FUNCTION_BLOCK Clearing_State  IMPLEMENTS ITF_State
VAR_INPUT
END_VAR
VAR_OUTPUT
END_VAR
VAR
	pPML_Base : POINTER TO PML_StatePattern_Base;
	_stateMachine : IPmlStateMachine;
END_VAR

METHOD Cycle : BOOL
_stateMachine.SetStateComplete();
pPML_Base^.SetState(pPML_Base^.stopped);
END_METHOD

METHOD FB_init : BOOL
VAR_INPUT
	bInitRetains : BOOL; // if TRUE, the retain variables are initialized (warm start / cold start)
	bInCopyCode : BOOL;  // if TRUE, the instance afterwards gets moved into the copy code (online change)
	pPML_Base : POINTER TO PML_StatePattern_Base;
	statemachine : IPmlStateMachine;
END_VAR
_stateMachine := statemachine;
THIS^.pPML_Base := pPML_Base;
END_METHOD

END_FUNCTION_BLOCK

(* stored: Version 1.1.0.1, ProductVersion 3.1.4024.12
   POU Clearing_State: Id {1f23ff1c-63dc-4572-a7ac-ed0a233c0084}, SpecialFunc None
   Method Cycle: Id {67af2511-d343-491e-9dbd-7f9fb6470886}
   Method FB_init: Id {7d0d3ea1-519d-47bd-aebe-ad8c7e3dea47} *)
